SUBAPPLICATION Softkey_Aux_Auto_IXA_TO_Remote_WRITE_BG_OPC (* VT-SoftKey lesen ODER AUX-Zuweisung (Joystick) lesen ODER lokaler Web-Override ODER Automatik-Kommando + Remote-OPC-UA-Write an Zielmodul + VT-Hintergrundfarbe (SoftKey UND AUX) aus Remote-Subscribe (generisch, ein Kanal). Kopie von Softkey_Aux_IXA_TO_Remote_WRITE_BG_OPC mit Softkey_Aux_Auto_IXA_TO_Remote_WRITE statt Softkey_Aux_IXA_TO_Remote_WRITE als Kommando-Haelfte - Status-Haelfte (AX_SUBSCRIBE_BG3_WEB_OPC) unveraendert. *)
  (* Standard: 61499-2 *)
  (* Version 1.1, 2026-09-16, Franz Höpfinger, Neuen WEB_STATE-Plug von Command durchgereicht (siehe Softkey_Aux_Auto_IXA_TO_Remote_WRITE Version 1.1) - behebt Doppel-Self-Subscribe, siehe BERICHT_2026-09-16_STG3_I1_I3_I4_I6_STALE_REMOTE_SUBSCRIBE.md Abschnitt 16-17. *)
  (* Version 1.0, 2026-09-11, Franz Höpfinger, Kopie von Softkey_Aux_IXA_TO_Remote_WRITE_BG_OPC (Version 1.2, 2026-09-07) mit Softkey_Aux_Auto_IXA_TO_Remote_WRITE als Kommando-Haelfte, fuer Achslenkung-Mittelpunkt-Automatik. *)
  PACKAGE MyLib::sys;
  (* Documentation:
  SoftKey UND Aux UND Automatik → Remote-OPC-UA-Write mit Status-Feedback (ein Kanal)
   Duennwandiger Wrapper, der Softkey_Aux_Auto_IXA_TO_Remote_WRITE (Kommando: SoftKey ODER Aux ODER lokaler Web-Override ODER Automatik → Remote-Write) und AX_SUBSCRIBE_BG3_WEB_OPC (Status: Remote-Subscribe → Hintergrundfarbe auf SoftKey UND Aux + lokaler Web-Republish, unveraendert) nebeneinanderstellt.
   Nur fuer Kanaele mit Automatik-Bedarf verwenden (aktuell: Achslenkung Links/Rechts, Hangausgleich Links/Rechts) - fuer alle anderen weiterhin Softkey_Aux_IXA_TO_Remote_WRITE_BG_OPC.
   WEB_STATE (neu, Version 1.1): durchgereichter Fan-out-Plug, siehe Softkey_Aux_Auto_IXA_TO_Remote_WRITE Version 1.1.
  *)
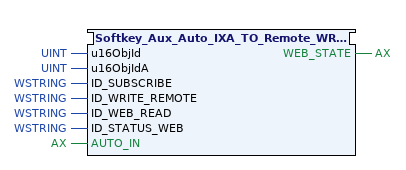
  VAR_INPUT
    u16ObjId : UINT; (* Object ID SoftKey/Hintergrund (VT) *)
    u16ObjIdA : UINT; (* Object ID AuxFunction2/Hintergrund (VT) *)
    ID_SUBSCRIBE : WSTRING; (* Remote-Subscribe-Adresse (Status/Farbe, ACTION=SUBSCRIBE) *)
    ID_WRITE_REMOTE : WSTRING; (* Remote-Write-Adresse zum Zielmodul (Befehl, ACTION=WRITE, CLIENT) *)
    ID_WEB_READ : WSTRING; (* Lokale Subscribe-Adresse fuer einen Web-Client (z.B. vt-ui-mirror) auf demselben Modul, ODER-verknuepft mit SoftKey und AUX *)
    ID_STATUS_WEB : WSTRING; (* Lokale Publish-Adresse (auf diesem Modul) fuer den vom Zielmodul zurueckgemeldeten Zustand - damit ein Web-Client (z.B. vt-ui-mirror) dieselbe Hintergrundfarbe wie das echte VT zeigen kann *)
  END_VAR
  SOCKETS
    AUTO_IN : adapter::types::unidirectional::AX; (* Autonomes Kommando (z.B. Achslenkung-Mittelpunkt-Automatik), ODER-verknuepft mit SoftKey/Aux/Web *)
  END_SOCKETS
  PLUGS
    WEB_STATE : adapter::types::unidirectional::AX; (* = Command.WEB_STATE durchgereicht, damit andere Composite-Instanzen denselben Web-Zustand ohne eigenen lokalen Self-Subscribe nutzen koennen *)
  END_PLUGS
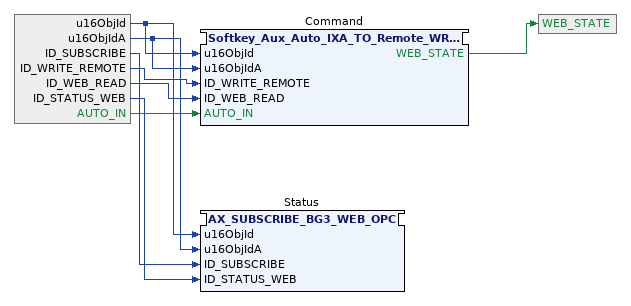
  SUBAPPS
    Command : MyLib::sys::Softkey_Aux_Auto_IXA_TO_Remote_WRITE;
    Status : MyLib::sys::AX_SUBSCRIBE_BG3_WEB_OPC;
  END_SUBAPPS
  DATA_CONNECTIONS
    u16ObjId TO Command.u16ObjId;
    u16ObjIdA TO Command.u16ObjIdA;
    ID_WRITE_REMOTE TO Command.ID_WRITE_REMOTE;
    ID_WEB_READ TO Command.ID_WEB_READ;
    u16ObjId TO Status.u16ObjId;
    u16ObjIdA TO Status.u16ObjIdA;
    ID_SUBSCRIBE TO Status.ID_SUBSCRIBE;
    ID_STATUS_WEB TO Status.ID_STATUS_WEB;
  END_CONNECTIONS
  ADAPTER_CONNECTIONS
    AUTO_IN TO Command.AUTO_IN;
    Command.WEB_STATE TO WEB_STATE;
  END_CONNECTIONS
END_SUBAPPLICATION
